// TIA Portal V19 export
DATA_BLOCK "time and date"   // DB89
{ S7_Optimized_Access := 'TRUE' }
// stored: MemoryReserve 100
   VAR RETAIN
      "Read time" : DTL;
      "write time" : DTL;
   END_VAR
   VAR
      "Set Time" : Bool;
      day : Int;
      month : Int;
      year : Int;
      hour : Int;
      minute : Int;
   END_VAR
   VAR RETAIN
      "Recipe Start Time" : DTL;
   END_VAR
BEGIN
END_DATA_BLOCK
